FUNCTION_BLOCK FB_Door
VAR_INPUT
	bInput			:	BOOL;	// Input über ein System
	bInputSwitch	:	BOOL;	// Input über einen Taster
	bInputPerm		:	BOOL;	// Input für dauerhaftes öffnen
	
	tPulse			:	TIME := T#5S;	//Zeit für High bei System oder HomeAssistant
	tPulseSwitch	:	TIME := tPulse;	//Zeit für High bei Schalter 
END_VAR
VAR_OUTPUT
	bOut			:	BOOL;
END_VAR
VAR_IN_OUT
	bInputHA		:	BOOL;	// Input über Home Assistant Taster
END_VAR
VAR CONSTANT
END_VAR
VAR
	fbRtrig			:	R_TRIG;
	fbRtrigSwitch	:	R_TRIG;
	fbRtrigHA		:	R_TRIG;
	
	tpPulse			:	TP;
	tpPulseSwitch	:	TP;
		
	bTrigger		:	BOOL;
	

	
END_VAR
VAR_TEMP

END_VAR

IF bInputPerm THEN
	
	bOut := TRUE;
	
ELSE

	bTrigger 	:= FALSE;

	fbRtrig(CLK:= bInput, Q=> );
	fbRtrigSwitch(CLK:= bInputSwitch, Q=> );
	fbRtrigHA(CLK:= bInputHA, Q=> );

	bTrigger := bTrigger OR fbRtrig.Q OR fbRtrigHA.Q;
	
	tpPulse(IN := bTrigger, PT := tPulse);
	tpPulseSwitch(IN := fbRtrigSwitch.Q, PT := tPulseSwitch);

	IF tpPulse.Q OR tpPulseSwitch.Q THEN
		bOut 		:= TRUE;
	ELSE
		bOut 		:= FALSE;
		bInputHA	:= FALSE;
	END_IF
	
END_IF

END_FUNCTION_BLOCK

(* stored: Version 1.1.0.1, ProductVersion 3.1.4024.4
   POU FB_Door: Id {1fb5dfc0-9653-43b7-a309-82bb47454417}, SpecialFunc None *)
